INTERFACE InterfaceJobEventObserver EXTENDS InterfaceObserverBase

METHOD OnError : BOOL
VAR_INPUT
	error_id : UDINT;
	message : STRING;
END_VAR
END_METHOD

METHOD OnJobEvent : BOOL
VAR_INPUT
	event : ST_JobEvent;
END_VAR
END_METHOD

END_INTERFACE

(* stored: Version 1.1.0.1, ProductVersion 3.1.4024.15
   Itf InterfaceJobEventObserver: Id {0ed931c1-423b-444d-b9d0-b8337c73de90}
   Method OnError: Id {99f8d7a2-4e81-4c8b-9a1c-2e8a4c7b8f64}
   Method OnJobEvent: Id {a8e6f3b4-7d52-4e9a-8c1b-5f2e9d8c7b6a} *)
